// TIA Portal V17 export
// export: Created 2024-09-02T12:49:57.2852075Z, ExportSetting WithDefaults, DisplayName Totally Integrated Automation Portal, DisplayVersion V17, DisplayName TIA Portal Openness, DisplayVersion V17, DisplayName TIA Portal Version Control Interface, DisplayVersion V17, DisplayName STEP 7 Professional, DisplayVersion V17, DisplayName STEP 7 Safety, DisplayVersion V17, DisplayName WinCC Professional, DisplayVersion V17
FUNCTION "HLP_BytetoBool" : Void   // FC30002, LAD
TITLE = Transfer Byte to Bool
{ S7_Optimized_Access := 'TRUE' }
AUTHOR : O.Fuehrus
FAMILY : HLP
NAME : HLP
VERSION : 1.0
// stored: AutoNumber false, IsIECCheckEnabled false, SetENOAutomatically false, UDAEnableTagReadback false
   VAR_INPUT
      iByte : Byte;
   END_VAR
   VAR_OUTPUT
      OUT0 : Bool;
      OUT1 : Bool;
      OUT2 : Bool;
      OUT3 : Bool;
      OUT4 : Bool;
      OUT5 : Bool;
      OUT6 : Bool;
      OUT7 : Bool;
   END_VAR
BEGIN

REGION Network 1
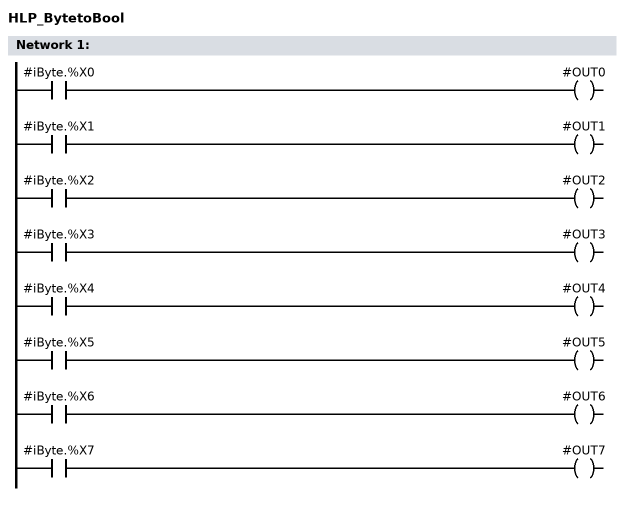
   RUNG wire#powerrail
      Contact( #iByte.%X0 )
      Coil( #OUT0 )
   END_RUNG
   RUNG wire#powerrail
      Contact( #iByte.%X1 )
      Coil( #OUT1 )
   END_RUNG
   RUNG wire#powerrail
      Contact( #iByte.%X2 )
      Coil( #OUT2 )
   END_RUNG
   RUNG wire#powerrail
      Contact( #iByte.%X3 )
      Coil( #OUT3 )
   END_RUNG
   RUNG wire#powerrail
      Contact( #iByte.%X4 )
      Coil( #OUT4 )
   END_RUNG
   RUNG wire#powerrail
      Contact( #iByte.%X5 )
      Coil( #OUT5 )
   END_RUNG
   RUNG wire#powerrail
      Contact( #iByte.%X6 )
      Coil( #OUT6 )
   END_RUNG
   RUNG wire#powerrail
      Contact( #iByte.%X7 )
      Coil( #OUT7 )
   END_RUNG
   // the same network as SCL:
   #OUT0 := #iByte.%X0;
   #OUT1 := #iByte.%X1;
   #OUT2 := #iByte.%X2;
   #OUT3 := #iByte.%X3;
   #OUT4 := #iByte.%X4;
   #OUT5 := #iByte.%X5;
   #OUT6 := #iByte.%X6;
   #OUT7 := #iByte.%X7;
END_REGION
END_FUNCTION
